TEXTLIST TextList_StationInfoPage
  1 = '1'
  2 = '2'
  3 = '3'
  4 = '4'
  5 = '5'
  6 = '6'
  10 = 'LOADING'
  11 = 'UNLOADING'
  13 = 'GENERAL'
   = ''
END_TEXTLIST

(* stored: Version 1.1.0.1, ProductVersion 3.1.4024.12
   TextList TextList_StationInfoPage: Id {e0865df5-6182-45f9-91eb-8d38734c997c} *)
